FUNCTION_BLOCK FB_Light IMPLEMENTS I_Switchable
VAR_OUTPUT
	// output of the FB. This is the state of the light.
	bActive AT %Q*: BOOL;
END_VAR

PROPERTY PUBLIC Active : BOOL
GET
Active := bActive;
END_GET
END_PROPERTY

METHOD Off : BOOL
bActive := false;
END_METHOD

METHOD On : BOOL
bActive := true;
END_METHOD

END_FUNCTION_BLOCK

(* stored: Version 1.1.0.1, ProductVersion 3.1.4024.5
   POU FB_Light: Id {c7346ac9-0c6b-4aa0-ae43-55b5f385f241}, SpecialFunc None
   Property Active: Id {2c31f253-24ee-413c-bec4-dadccd1ea919}
   Get Get: Id {3c7b4bb3-6c5e-4e93-93a3-84dc12254a48}
   Method Off: Id {352e17f0-b85c-42a2-b903-34ea7807ce68}
   Method On: Id {69bbc1b6-42ee-45ce-a690-92d654fbb732} *)
